(* CoDeSys 2.3.9.41 project: Блок управления светофором.pro *)
(* Libraries: Standard.lib 4.10.05 11:14:46, IecSfc.lib 13.4.06 15:51:28, SYSLIBCALLBACK.LIB 26.9.08 16:43:52 *)

(* Global variable list: Global_Variables *)
VAR_GLOBAL
	IN:BOOL;
	L1_GREEN:BOOL;
	L1_YELLOW:BOOL;
	L1_RED:BOOL;
	L2_GREEN:BOOL;
	L2_YELLOW:BOOL;
	L2_RED:BOOL;
END_VAR

(* POU PLC_PRG, CFC *)
PROGRAM PLC_PRG
VAR
	LIGHT1: TRAFFICSIGNAL;
	LIGHT2: TRAFFICSIGNAL;
	END_VAR
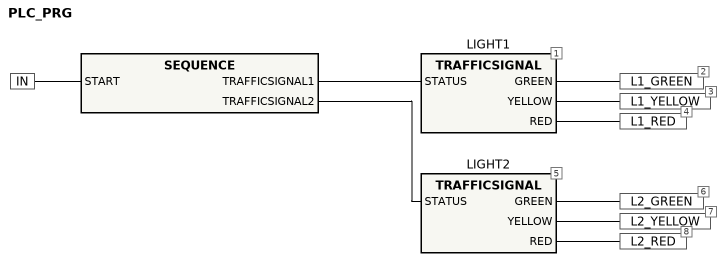
_CFC_ (* Continuous Function Chart, elements in execution order *)
#0 SEQUENCE(START: IN)
#1 LIGHT1:TRAFFICSIGNAL(STATUS: #0.TRAFFICSIGNAL1)
#2 L1_GREEN <= #1.GREEN
#3 L1_YELLOW <= #1.YELLOW
#4 L1_RED <= #1.RED
#5 LIGHT2:TRAFFICSIGNAL(STATUS: #0.TRAFFICSIGNAL2)
#6 L2_GREEN <= #5.GREEN
#7 L2_YELLOW <= #5.YELLOW
#8 L2_RED <= #5.RED
_END_CFC_
(* the same logic as Structured Text *)
SEQUENCE(START := IN);
LIGHT1(STATUS := SEQUENCE.TRAFFICSIGNAL1);
L1_GREEN := LIGHT1.GREEN;
L1_YELLOW := LIGHT1.YELLOW;
L1_RED := LIGHT1.RED;
LIGHT2(STATUS := SEQUENCE.TRAFFICSIGNAL2);
L2_GREEN := LIGHT2.GREEN;
L2_YELLOW := LIGHT2.YELLOW;
L2_RED := LIGHT2.RED;
END_PROGRAM

(* POU TRAFFICSIGNAL, FBD *)
FUNCTION_BLOCK TRAFFICSIGNAL
VAR_INPUT
	STATUS: INT;
END_VAR
VAR_OUTPUT
	GREEN: BOOL;
	YELLOW: BOOL;
	RED: BOOL;
END_VAR
VAR
	OFF:BOOL;
END_VAR
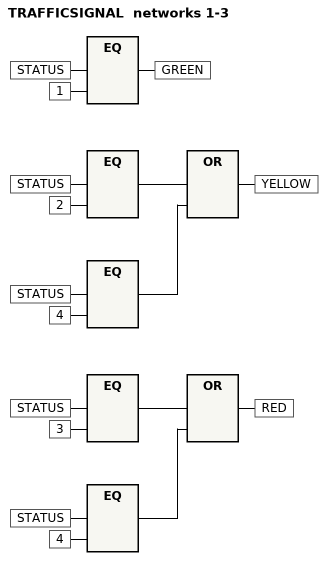
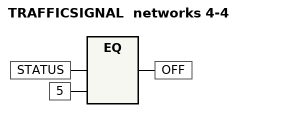
_FBD_ (* Function Block Diagram *)
NETWORK 1
	EQ(STATUS, 1) => GREEN
NETWORK 2
	OR(EQ(STATUS, 2), EQ(STATUS, 4)) => YELLOW
NETWORK 3
	OR(EQ(STATUS, 3), EQ(STATUS, 4)) => RED
NETWORK 4
	EQ(STATUS, 5) => OFF
_END_FBD_
(* the same logic as Structured Text *)
(* Network 1 *)
GREEN := STATUS = 1;
(* Network 2 *)
YELLOW := (STATUS = 2) OR (STATUS = 4);
(* Network 3 *)
RED := (STATUS = 3) OR (STATUS = 4);
(* Network 4 *)
OFF := STATUS = 5;
END_FUNCTION_BLOCK

(* POU SEQUENCE, SFC *)
PROGRAM SEQUENCE

VAR_INPUT
	START: BOOL;
END_VAR
VAR_OUTPUT
	TRAFFICSIGNAL1: INT;
	TRAFFICSIGNAL2: INT;
END_VAR
VAR
	COUNTER:INT;
	DELAY: WAIT;
END_VAR
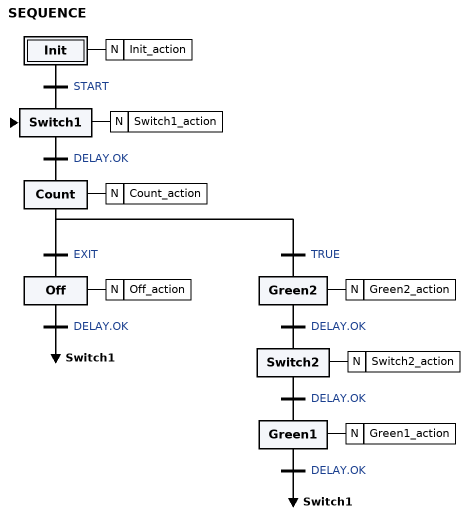
INITIAL_STEP Init:
	Init_action(N);
END_STEP
TRANSITION FROM Init TO Switch1 := START;
END_TRANSITION
STEP Switch1:
	Switch1_action(N);
END_STEP
TRANSITION FROM Switch1 TO Count := DELAY.OK;
END_TRANSITION
STEP Count:
	Count_action(N);
END_STEP
TRANSITION FROM Count TO Off := EXIT;
END_TRANSITION
TRANSITION FROM Count TO Green2 := TRUE;
END_TRANSITION
STEP Off:
	Off_action(N);
END_STEP
TRANSITION FROM Off TO Switch1 := DELAY.OK;
END_TRANSITION
STEP Green2:
	Green2_action(N);
END_STEP
TRANSITION FROM Green2 TO Switch2 := DELAY.OK;
END_TRANSITION
STEP Switch2:
	Switch2_action(N);
END_STEP
TRANSITION FROM Switch2 TO Green1 := DELAY.OK;
END_TRANSITION
STEP Green1:
	Green1_action(N);
END_STEP
TRANSITION FROM Green1 TO Switch1 := DELAY.OK;
END_TRANSITION

ACTION Init_action:
	LD		1
	ST		TRAFFICSIGNAL1
	LD		3
	ST		TRAFFICSIGNAL2
END_ACTION

ACTION Switch1_action:
	LD		2
	ST		TRAFFICSIGNAL1
	LD		4
	ST		TRAFFICSIGNAL2
	CAL		DELAY(TIME_IN:=t#2s)
END_ACTION

ACTION Count_action:
	LD		COUNTER
	ADD		1
	ST		COUNTER
END_ACTION

ACTION Off_action:
	LD		5
	ST		TRAFFICSIGNAL1
	LD		5
	ST		TRAFFICSIGNAL2
	LD		0
	ST		COUNTER
	CAL		DELAY(TIME_IN:=t#10s)
END_ACTION

ACTION Green2_action:
	LD		3
	ST		TRAFFICSIGNAL1
	LD		1
	ST		TRAFFICSIGNAL2
	CAL		DELAY(TIME_IN:=t#5s)
END_ACTION

ACTION Switch2_action:
	LD		4
	ST		TRAFFICSIGNAL1
	LD		2
	ST		TRAFFICSIGNAL2
	CAL		DELAY(TIME_IN:=t#2s)
END_ACTION

ACTION Green1_action:
	LD		1
	ST		TRAFFICSIGNAL1
	LD		3
	ST		TRAFFICSIGNAL2
	CAL		DELAY(TIME_IN:=t#5s)
END_ACTION

TRANSITION EXIT:
	LD		COUNTER
	GT		7
END_TRANSITION
END_PROGRAM

(* POU WAIT, IL *)
FUNCTION_BLOCK WAIT
VAR_INPUT
	TIME_IN: TIME;
END_VAR
VAR_OUTPUT
	OK: BOOL := FALSE;
END_VAR
VAR
	ZAB:TP;
END_VAR
	LD		ZAB.Q
	JMPC	mark

	CAL		ZAB(IN:=FALSE)
	LD		TIME_IN
	ST		ZAB.PT
	CAL		ZAB(IN:=TRUE)
	JMP		end

mark:
	CAL		ZAB
end:
	LDN		ZAB.Q
	ST		OK
	RET
END_FUNCTION_BLOCK

(* Visualisation lights
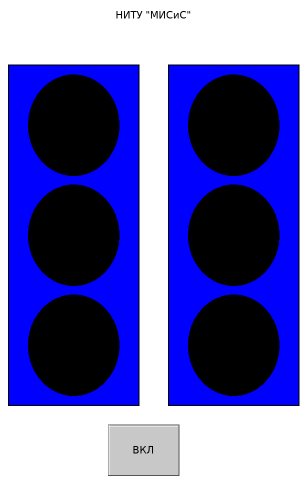
ellipse at (190,340)-(281,441): alarm colour if .L1_GREEN
ellipse at (190,230)-(281,331): alarm colour if .L1_YELLOW
ellipse at (190,120)-(281,221): alarm colour if .L1_RED
ellipse at (350,340)-(441,441): alarm colour if .L2_GREEN
ellipse at (350,230)-(441,331): alarm colour if .L2_YELLOW
ellipse at (350,120)-(441,221): alarm colour if .L2_RED
button at (270,470)-(341,521): text "ВКЛ"; taps .IN
rounded rectangle at (140,30)-(491,91): text "НИТУ "МИСиС""
2 more shapes without text or variables
*)
